Staubli VAL3: getItem.pgx

public program getItem(InstrItem& x_sItem, num x_nIndex)
begin
  // give back the instruction
  x_sItem=pEdit.iEvent[x_nIndex]
end
